(* IEC 61131-3 sources: ArfBotOS/Codesys-4/ArfBotOS.fbsdev/Application.iecapp^/FUN/digital/FB_DigitalOutput.fb.st^/P_StateOn.prop.st^, 1 file *)

(* ---- Get.meth.st ---- *)
VAR
END_VAR

P_StateOn := _Output;
